// SIMATIC S7-200 SMART project (STEP 7-Micro/WIN SMART), CPU SR20

SYMBOL_TABLE System Symbols
Always_On        SM0.0    // Always ON
END_SYMBOL_TABLE

ORGANIZATION_BLOCK MAIN:OB1
TITLE=Program Comments
BEGIN
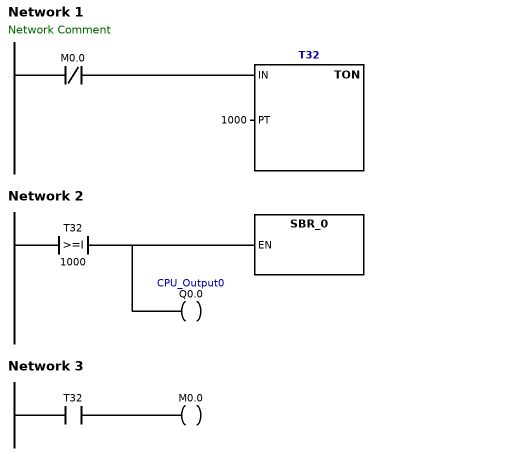
Network 1
// Network Comment
LDN    M0.0
TON    T32, 1000
Network 2
LDW>=  T32, 1000
CALL   SBR_0:SBR0
=      CPU_Output0:Q0.0
Network 3
LD     T32
=      M0.0
END_ORGANIZATION_BLOCK

SUBROUTINE_BLOCK SBR_0:SBR0
TITLE=Subroutine Comments
BEGIN
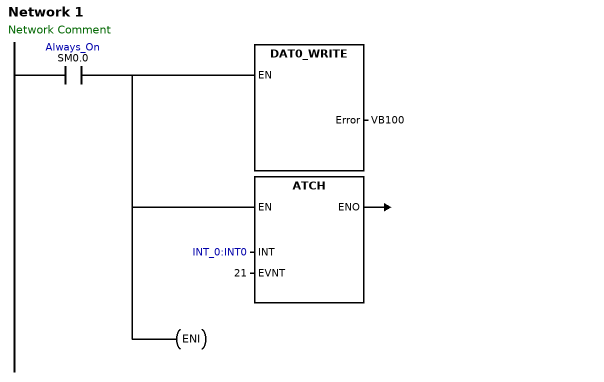
Network 1
// Network Comment
LD     Always_On:SM0.0
CALL   DAT0_WRITE:SBR1, VB100
ATCH   INT_0:INT0, 21
ENI
END_SUBROUTINE_BLOCK

// SBR1: protected block, not included

INTERRUPT_BLOCK INT_0:INT0
TITLE=Interrupt routine comments
BEGIN
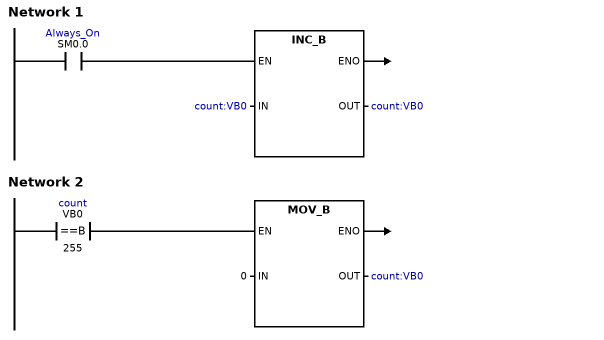
Network 1
LD     Always_On:SM0.0
INCB   count:VB0
Network 2
LDB=   count:VB0, 255
MOVB   0, count:VB0
END_INTERRUPT_BLOCK
